Fanuc KAREL source: kb00127.KL

-- PROVISIONAL review KL for V940-1; original PC SHA256 625de6d51ed18760350538c8602de8c85460151662ef34fadeadf4261faad9d7
-- Incomplete behavior may be omitted. Consult companion uncertainty JSON. Do not deploy.
PROGRAM KB00127
%NOLOCKGROUP
VAR
  P1 : STRING[80]
  P2 : INTEGER
  RESULT : INTEGER
BEGIN
  -- V9_ZERO_TABLE_METADATA_HINT layout=0001; no indexed target words; source/name/runtime held
  -- UNRESOLVED_PC offsets 5-14; opcodes 3F,75
  -- UNRESOLVED_PC offsets 19-26; opcodes 9D,23
  -- UNRESOLVED_PC offsets 31-54; opcodes 27,22,2A,22,76,23
  -- UNRESOLVED_PC offsets 59-63; opcodes 7F
END KB00127
